PROGRAM MAIN
VAR
END_VAR

END_PROGRAM

(* stored: Version 1.1.0.1
   POU MAIN: Id {c4659204-b884-47e8-bf67-3e6c4766ddfe} *)
